// TIA Portal V20 export
VAR_GLOBAL   // PLC tag table "LNK_Const_Rt"
END_VAR
VAR_GLOBAL CONSTANT   // user constants
   LNK_ROLE_ACTIVE : USInt := 1;   // Link role: PLC opens the TCP connection (client) / 링크 역할: PLC 가 연결 (클라이언트)
   LNK_ROLE_PASSIVE : USInt := 2;   // Link role: PLC listens for one peer (server) / 링크 역할: PLC 가 대기 (서버, 단일 피어)
   LNK_FRM_FRAME : USInt := 1;   // Framing: 16-byte header + payload / 프레이밍: 16 B 헤더 + 페이로드
   LNK_FRM_HTTP : USInt := 2;   // Framing: HTTP/1.1 subset / 프레이밍: HTTP/1.1 (부분 집합)
   LNK_FRM_NDJSON : USInt := 3;   // Framing: one JSON envelope per line (JSON only) / 프레이밍: 줄 단위 JSON 엔벨로프 (JSON 전용)
   LNK_ST_DISABLED : USInt := 0;   // Connection state: slot disabled (FB_LnkConn Enable FALSE) / 연결 상태: 슬롯 비활성
   LNK_ST_IDLE : USInt := 1;   // Connection state: enabled, waiting for instructions to be free before TCON / 연결 상태: 사용, TCON 전 명령어 BUSY 해제 대기
   LNK_ST_CONNECTING : USInt := 2;   // Connection state: TCON running (connecting / listening) / 연결 상태: TCON 진행 (연결 중 / 대기)
   LNK_ST_UP : USInt := 3;   // Connection state: established / 연결 상태: 연결됨
   LNK_ST_CLOSING : USInt := 4;   // Connection state: TDISCON running / 연결 상태: 연결 해제 중
   LNK_ST_BACKOFF : USInt := 5;   // Connection state: waiting before reconnect (1-2-4 s) / 연결 상태: 재접속 대기 (1-2-4 s)
   LNK_PH_IDLE : USInt := 0;   // Command inject phase: idle / 명령 주입 단계: 없음
   LNK_PH_INJECTED : USInt := 1;   // Command inject phase: injected, restore next cycle / 명령 주입 단계: 주입됨, 다음 사이클 복원
   LNK_RX_LAST : DInt := 8191;   // Receive accumulation buffer last index (RxBuf[0..8191]) / 수신 누적 버퍼 마지막 인덱스 (RxBuf[0..8191])
   LNK_CHUNK_LAST : DInt := 1459;   // TRCV ad-hoc chunk buffer last index (1460 B) / TRCV ADHOC 1 회 수신 버퍼 마지막 인덱스 (1460 B)
   LNK_MSGBUF_LAST : DInt := 8192;   // Message buffer last index (8192 B + 0 terminator) / 메시지 버퍼 마지막 인덱스 (8192 B + 0 종단)
   LNK_TX_LAST : DInt := 8191;   // Transmit buffer last index (TxBuf[0..8191]) / 송신 버퍼 마지막 인덱스 (TxBuf[0..8191])
   LNK_HTTP_HDR_MAX : DInt := 1024;   // HTTP header section max bytes on the PLC (else 431) / PLC HTTP 헤더 섹션 최대 바이트 (초과 시 431)
   LNK_CONNID_1 : Word := 16#0120;   // Connection ID of link slot 1 / 링크 슬롯 1 연결 ID
   LNK_CONNID_2 : Word := 16#0121;   // Connection ID of link slot 2 / 링크 슬롯 2 연결 ID
   LNK_HTTP_GET : USInt := 1;   // HTTP method GET / HTTP 메서드 GET
   LNK_HTTP_POST : USInt := 2;   // HTTP method POST / HTTP 메서드 POST
   LNK_RT_NONE : USInt := 0;   // HTTP route: none / unknown path / HTTP 경로: 없음 / 알 수 없음
   LNK_RT_COMMAND : USInt := 1;   // HTTP route (PLC passive): POST /api/command / HTTP 경로 (PLC Passive): POST /api/command
   LNK_RT_STATUS : USInt := 2;   // HTTP route (PLC passive): GET /api/status / HTTP 경로 (PLC Passive): GET /api/status
   LNK_RT_MEASLOG_LAST : USInt := 3;   // HTTP route (PLC passive): GET /api/measlog/last / HTTP 경로 (PLC Passive): GET /api/measlog/last
   LNK_RT_HELLO : USInt := 4;   // HTTP route (PLC passive): GET /api/hello / HTTP 경로 (PLC Passive): GET /api/hello
   LNK_RT_PLC_MSG : USInt := 10;   // HTTP route (PC server): POST /api/plc/<Plc>/<msg> / HTTP 경로 (PC 서버): POST /api/plc/<Plc>/<msg>
   LNK_RT_PLC_COMMAND : USInt := 11;   // HTTP route (PC server): GET /api/plc/<Plc>/command / HTTP 경로 (PC 서버): GET /api/plc/<Plc>/command
   LNK_E_CMD_DISABLED : Int := 100;   // Command rejected: CmdEnable / AcceptCommand off / 명령 거부: CmdEnable / AcceptCommand 꺼짐
   LNK_E_CMD_HEADER : Int := 101;   // Command rejected: header zero / no command / 명령 거부: 헤더 0 / 명령 없음
   LNK_E_CMD_SRC : Int := 102;   // Command rejected: SRC is GRM (4000) / 명령 거부: SRC 가 GRM (4000)
   LNK_E_CMD_DST : Int := 103;   // Command rejected: DST is not this machine / 명령 거부: DST 가 이 설비 ID 아님
   LNK_E_CMD_UNSUPPORTED : Int := 104;   // Command rejected: Jog / B3 / Home / MaintPos / CellOrigin not supported / 명령 거부: Jog / B3 / Home / MaintPos / CellOrigin 미지원
   LNK_E_CMD_MASKED : Int := 105;   // Command rejected: Reset / Initializing / ChangeMode without AllowManual / 명령 거부: AllowManual 없이 Reset / Initializing / ChangeMode
   LNK_E_CMD_WAIT : Int := 106;   // Command not injected this cycle (session retries, BUSY after CmdWaitMs) / 명령 이번 사이클 주입 불가 (세션 재시도, CmdWaitMs 초과 시 BUSY)
   LNK_E_TCON : Int := 200;   // Transport error: TCON failed / 전송 오류: TCON 실패
   LNK_E_TDISCON : Int := 201;   // Transport error: TDISCON failed / 전송 오류: TDISCON 실패
   LNK_E_TSEND : Int := 202;   // Transport error: TSEND failed / 전송 오류: TSEND 실패
   LNK_E_TRCV : Int := 203;   // Transport error: TRCV failed / 전송 오류: TRCV 실패
   LNK_E_CONN_TIMEOUT : Int := 204;   // Transport error: connect timeout (active) / 전송 오류: 연결 시간 초과 (Active)
   LNK_E_PEER_CLOSED : Int := 205;   // Transport error: peer closed the connection / 전송 오류: 피어가 연결 종료
   LNK_E_RX_OVERFLOW : Int := 206;   // Transport error: receive buffer full without a complete message / 전송 오류: 완전한 메시지 없이 수신 버퍼 가득
   LNK_E_HB_TIMEOUT : Int := 207;   // Transport error: nothing received for 3 x HeartbeatMs / 전송 오류: 3 x HeartbeatMs 동안 무수신
   LNK_JERR_OVERFLOW : DInt := -5;   // Json/Frame writer sticky error in Pos: buffer overflow / Json/Frame 쓰기 끈끈한 오류 (Pos): 버퍼 넘침
   LNK_JERR_PARSE : DInt := -6;   // Json/Frame reader sticky error in Pos: syntax / range / Json/Frame 읽기 끈끈한 오류 (Pos): 문법 / 범위
   LNK_TRACE_CH_MAX : Int := 32;   // Trace: maximum channels (LNK_TraceCfg.Chan upper bound + 1)
   LNK_TRACE_WORDS : Int := 2032;   // Trace: DWord elements of one chunk (LNK_Trace.Data)
   LNK_TRACE_CHUNK_LAST : Int := 3;   // Trace: upper bound of the chunk ring (TRACE_LNK.Chunk)
   LNK_TRACE_FLUSH_MIN : UInt := 20;   // Trace: smallest accepted FlushMs (ms)
   LNK_PEEK_I : Byte := 16#81;   // PEEK area: process image input
   LNK_PEEK_Q : Byte := 16#82;   // PEEK area: process image output
   LNK_PEEK_M : Byte := 16#83;   // PEEK area: bit memory
   LNK_PEEK_DB : Byte := 16#84;   // PEEK area: data block (standard access only)
   LNK_E_TRACE_CFG : Int := 110;   // Trace: rejected TraceCfg (channel, width, area or timing invalid)
   LNK_E_TRACE_OFF : Int := 111;   // Trace: not allowed on this slot (AllowTrace FALSE or framing is not FRAME)
END_VAR
